FUNCTION_BLOCK Pallet
  (* Standard: 61499-2 *)
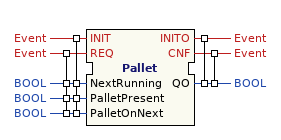
  EVENT_INPUT
    INIT WITH NextRunning, PalletPresent, PalletOnNext;
    REQ WITH NextRunning, PalletPresent, PalletOnNext;
  END_EVENT
  EVENT_OUTPUT
    INITO WITH QO;
    CNF WITH QO;
  END_EVENT
  VAR_INPUT
    NextRunning : BOOL;
    PalletPresent : BOOL;
    PalletOnNext : BOOL;
  END_VAR
  VAR_OUTPUT
    QO : BOOL;
  END_VAR
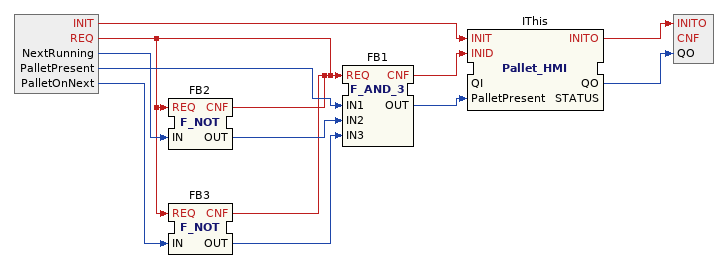
  FBS
    IThis : Pallet_HMI;
    FB1 : F_AND_3;
    FB2 : F_NOT;
    FB3 : F_NOT;
  END_FBS
  EVENT_CONNECTIONS
    REQ TO FB2.REQ;
    INIT TO IThis.INIT;
    IThis.INITO TO INITO;
    REQ TO FB1.REQ;
    FB2.CNF TO FB1.REQ;
    FB1.CNF TO IThis.INID;
    REQ TO FB3.REQ;
    FB3.CNF TO FB1.REQ;
  END_CONNECTIONS
  DATA_CONNECTIONS
    NextRunning TO FB2.IN;
    IThis.QO TO QO;
    PalletPresent TO FB1.IN1;
    FB2.OUT TO FB1.IN2;
    FB1.OUT TO IThis.PalletPresent;
    FB3.OUT TO FB1.IN3;
    PalletOnNext TO FB3.IN;
  END_CONNECTIONS
END_FUNCTION_BLOCK
